{attribute 'Tc2GvlVarNames'}
VAR_GLOBAL
	Defaut_Bus_de_Terrain:BOOL:=FALSE;

	State_Maitre_Ethercat_Visu		:INT;

END_VAR

(* stored: Version 1.1.0.1
   GVL Global_Ethercat: Id {34d1d07c-c5a3-4009-87a4-459fbdf2e2fe} *)
